# EPICS substitutions: iocBoot/ioc13bmc/Pelco_CM6700.substitutions
file "$(IP)/ipApp/Db/Pelco_CM6700.db"
{
pattern
{P,       R,       PORT}
{13BMC:,  Pelco1,  serial7}
}

file "$(IP)/ipApp/Db/Pelco_CM6700_names.db"
{
pattern
{P,       R,       STR}
{13BMC:,  Pelco1,  ZRST}
{13BMC:,  Pelco1,  ONST}
{13BMC:,  Pelco1,  TWST}
{13BMC:,  Pelco1,  THST}
{13BMC:,  Pelco1,  FRST}
{13BMC:,  Pelco1,  FVST}
{13BMC:,  Pelco1,  SXST}
{13BMC:,  Pelco1,  SVST}
{13BMC:,  Pelco1,  EIST}
{13BMC:,  Pelco1,  NIST}
{13BMC:,  Pelco1,  TEST}
{13BMC:,  Pelco1,  ELST}
{13BMC:,  Pelco1,  TVST}
{13BMC:,  Pelco1,  TTST}
{13BMC:,  Pelco1,  FTST}
{13BMC:,  Pelco1,  FFST}
}
